INTERFACE LightTower

METHOD Blink : BOOL
VAR_INPUT
	On : BOOL;
END_VAR
END_METHOD

METHOD OnOff
VAR_INPUT
	On : BOOL;
END_VAR
END_METHOD

END_INTERFACE

(* stored: Version 1.1.0.1, ProductVersion 3.1.4024.12
   Itf LightTower: Id {f2fc1df0-adb7-4881-8fa2-74376db605ce}
   Method Blink: Id {579309b6-9baf-4cc1-8024-191493ee0057}
   Method OnOff: Id {527154b4-46d6-474e-be8b-e54abe4d77df} *)
